{attribute addProperty BoxType "EK1100-0000-0018"}
{attribute addProperty Id "Beckhoff_ER8xxxEK1122Beckhoff_ER8xxxEK1122_05C4D0D141051.25"}
{attribute addProperty CRC "3167703383"}
{attribute addProperty SizeInBites "410"}
{attribute addProperty SizeInBytes "51.25"}
TYPE Beckhoff_ER8xxx_BCCF5157 EXTENDS EK1100_179A0949 :
STRUCT
	{attribute addProperty Name "Beckhoff_ER8xxxEK1122"}
	Beckhoff_ER8xxxEK1122 : Beckhoff_ER8xxxEK1122_05C4D0D1;
END_STRUCT
END_TYPE

(* stored: Version 1.2.0.0, ProductVersion 3.1.4024.9
   DUT Beckhoff_ER8xxx_BCCF5157: Id {d680e317-033d-4d59-ae81-f98079a4d6af} *)
